{attribute 'qualified_only'}
VAR_GLOBAL CONSTANT
    DP_ID_DEFAULT_DATATYPE                   : UINT := 16#0000;
    DP_ID_PP_EMERGENCY_2                     : UINT := 16#0003;
    DP_ID_PP_EMERGENCY_1                     : UINT := 16#0004;

    DP_ID_DEBUG                              : UINT := 16#0069;
    DP_ID_MAIN_PCB_BOOT                      : UINT := 16#0070;

    DP_ID_COMMAND_HASH                       : UINT := 16#0167;
    DP_ID_DATA_HASH                          : UINT := 16#0169;
    DP_ID_VALUE_ERROR                        : UINT := 16#016A;
    DP_ID_VALUE_WARNING                      : UINT := 16#016B;
    DP_ID_VALUE_CAUSED_BRAKING               : UINT := 16#016C;
    DP_ID_LOCALISATION_HEARTBEAT             : UINT := 16#016E;
    DP_ID_SENSOR_HUB_HEARTBEAT               : UINT := 16#016F;
    DP_ID_FRONTEND_HEARTBEATING              : UINT := 16#0170;
    DP_ID_CONFIG_HASH                        : UINT := 16#0171;

    DP_ID_HV_V_LOW                           : UINT := 16#019D;   // critical
    DP_ID_BMS_TEMPERATURE_LOW                : UINT := 16#019E;

    DP_ID_FSM_STATE                          : UINT := 16#0202;
    DP_ID_FSM_TRANSITION_FAIL                : UINT := 16#0204;
    DP_ID_EMERGENCY                          : UINT := 16#0205;

    DP_ID_LEVI_SYSTEM_CHECK_SUCCESS          : UINT := 16#0220;
    DP_ID_LEVI_SYSTEM_CHECK_FAILURE          : UINT := 16#0221;
    DP_ID_PROP_1_SYSTEM_CHECK_SUCCESS        : UINT := 16#0222;
    DP_ID_PROP_1_SYSTEM_CHECK_FAILURE        : UINT := 16#0223;
    DP_ID_PROP_2_SYSTEM_CHECK_SUCCESS        : UINT := 16#0224;
    DP_ID_PROP_2_SYSTEM_CHECK_FAILURE        : UINT := 16#0225;
    DP_ID_RESET_FSM                          : UINT := 16#0226;
    DP_ID_EMERGENCY_STALE_CRITICAL_DATA      : UINT := 16#0227;
    DP_ID_LOCALIZATION_LIMIT_REACHED         : UINT := 16#0228;

    DP_ID_POD_STATE                          : UINT := 16#0250;   // u16,  pod->gs,  critical
    DP_ID_EMERGENCY_REASON                   : UINT := 16#0251;   // u16,  bidir,  critical
    DP_ID_POD_STATE_COMMAND                  : UINT := 16#0252;   // u16,  gs->pod

    DP_ID_LOCALIZATION                       : UINT := 16#0321;   // f32,  mm,  pod->gs

    DP_ID_HV_V_HIGH                          : UINT := 16#03A1;   // critical
    DP_ID_BMS_TEMPERATURE_HIGH               : UINT := 16#03A2;
    DP_ID_HVAL_STATE                         : UINT := 16#03A4;
    DP_ID_VDC_LINK                           : UINT := 16#03A7;   // critical
    DP_ID_PTC_ERRORS                         : UINT := 16#03B1;

    DP_ID_TEMP_MOTOR_LEFT_0                  : UINT := 16#04B0;
    DP_ID_TEMP_MOTOR_LEFT_1                  : UINT := 16#04B1;
    DP_ID_TEMP_MOTOR_LEFT_2                  : UINT := 16#04B2;
    DP_ID_TEMP_MOTOR_LEFT_3                  : UINT := 16#04B3;
    DP_ID_TEMP_MOTOR_LEFT_4                  : UINT := 16#04B4;
    DP_ID_TEMP_MOTOR_LEFT_5                  : UINT := 16#04B5;
    DP_ID_WORD_2                             : UINT := 16#04B6;   // critical
    DP_ID_IBUS_1                             : UINT := 16#04C2;
    DP_ID_IBUS_2                             : UINT := 16#04C6;

    DP_ID_PP_INIT_FAULT_1                    : UINT := 16#0507;
    DP_ID_PP_INIT_FAULT_2                    : UINT := 16#0508;
    DP_ID_TEMP_MOTOR_RIGHT_1                 : UINT := 16#050A;
    DP_ID_TEMP_MOTOR_RIGHT_2                 : UINT := 16#050B;
    DP_ID_TEMP_MOTOR_RIGHT_3                 : UINT := 16#050C;
    DP_ID_TEMP_MOTOR_RIGHT_4                 : UINT := 16#050D;
    DP_ID_TEMP_MOTOR_RIGHT_5                 : UINT := 16#050E;
    DP_ID_TEMP_MOTOR_RIGHT_6                 : UINT := 16#050F;

    DP_ID_TEMP_MOTOR_RIGHT_0                 : UINT := 16#0520;
    DP_ID_VELOCITY                           : UINT := 16#0527;   // i16,  mm/s,  pod->gs
    DP_ID_ROLL                               : UINT := 16#052E;
    DP_ID_PITCH                              : UINT := 16#052F;
    DP_ID_YAW                                : UINT := 16#0530;
    DP_ID_TEMP_HEMS1                         : UINT := 16#053C;
    DP_ID_TEMP_HEMS2                         : UINT := 16#053D;
    DP_ID_TEMP_HEMS3                         : UINT := 16#053E;
    DP_ID_TEMP_HEMS4                         : UINT := 16#053F;
    DP_ID_TEMP_HEMS5                         : UINT := 16#0540;
    DP_ID_TEMP_HEMS6                         : UINT := 16#0541;
    DP_ID_TEMP_HEMS7                         : UINT := 16#0542;
    DP_ID_TEMP_HEMS8                         : UINT := 16#0543;
    DP_ID_TEMP_EMS1                          : UINT := 16#0544;
    DP_ID_TEMP_EMS2                          : UINT := 16#0545;
    DP_ID_TEMP_EMS3                          : UINT := 16#0546;
    DP_ID_TEMP_EMS4                          : UINT := 16#0547;
    DP_ID_TEMP_EMS5                          : UINT := 16#0548;
    DP_ID_TEMP_EMS6                          : UINT := 16#0549;
    DP_ID_TEMP_EMS7                          : UINT := 16#054A;
    DP_ID_TEMP_EMS8                          : UINT := 16#054B;
    DP_ID_TEMP_MOTOR_RIGHT_7                 : UINT := 16#0555;
    DP_ID_TEMP_MOTOR_LEFT_6                  : UINT := 16#0556;
    DP_ID_TEMP_MOTOR_LEFT_7                  : UINT := 16#0557;
    DP_ID_LEVI_HEARTBEAT                     : UINT := 16#0567;   // critical
    DP_ID_LEVI_FAULT                         : UINT := 16#0568;

    DP_ID_WORD_1                             : UINT := 16#05B8;   // critical

    DP_ID_ISOLATION_RESISTANCE               : UINT := 16#0610;   // critical
    DP_ID_BUS_CURRENT                        : UINT := 16#0611;   // critical

    DP_ID_PRESSURE_LOW                       : UINT := 16#0666;   // critical
    DP_ID_PRESSURE_HIGH                      : UINT := 16#0667;   // critical

    DP_ID_SENSOR_HUB_EMERGENCY               : UINT := 16#0696;
    DP_ID_PTC_ERROR_EMERGENCY                : UINT := 16#0697;
    DP_ID_BMS_ERROR_LOW_VOLTAGE              : UINT := 16#0698;
    DP_ID_BMS_ERROR_HIGH_VOLTAGE             : UINT := 16#0699;

    DP_ID_LEVI_FAULT_DRIVE_NUMBER            : UINT := 16#0777;

    DP_ID_OFFSET_1                           : UINT := 16#0848;   // f32,  mm,  pod->gs
    DP_ID_OFFSET_2                           : UINT := 16#0849;   // f32,  mm,  pod->gs
    DP_ID_OFFSET_3                           : UINT := 16#084A;   // f32,  mm,  pod->gs
    DP_ID_OFFSET_4                           : UINT := 16#084B;   // f32,  mm,  pod->gs
    DP_ID_OFFSET_5                           : UINT := 16#084C;   // f32,  mm,  pod->gs
    DP_ID_OFFSET_6                           : UINT := 16#084D;   // f32,  mm,  pod->gs

    DP_ID_BARCODE_POSITION                   : UINT := 16#0900;
    DP_ID_BARCODE_VELOCITY                   : UINT := 16#0901;
    DP_ID_BARCODE_ID                         : UINT := 16#0902;
    DP_ID_BARCODE_QUALITY                    : UINT := 16#0903;
    DP_ID_LEVI_STATE                         : UINT := 16#0904;   // i16,  pod->gs,  critical
    DP_ID_LEVI_COMMAND                       : UINT := 16#0905;   // i16,  bidir,  critical
    DP_ID_LEVI_READY                         : UINT := 16#0906;   // u8,  pod->gs
    DP_ID_LEVI_Z_TARGET                      : UINT := 16#0907;   // f64,  m,  pod->gs
    DP_ID_LEVI_PITCH_TARGET                  : UINT := 16#0908;   // f64,  rad,  pod->gs
    DP_ID_LEVI_ROLL_TARGET                   : UINT := 16#0909;   // f64,  rad,  pod->gs
    DP_ID_LEVI_Y_TARGET_AIRGAP               : UINT := 16#090A;   // f64,  m,  pod->gs
    DP_ID_LEVI_YAW_TARGET                    : UINT := 16#090B;   // f64,  rad,  pod->gs
    DP_ID_LEVI_Z_LIFTOFF                     : UINT := 16#090C;   // f64,  m,  pod->gs
    DP_ID_LEVI_Z                             : UINT := 16#090D;   // f64,  m,  pod->gs,  critical
    DP_ID_LEVI_ROLL                          : UINT := 16#090E;   // f64,  rad,  pod->gs,  critical
    DP_ID_LEVI_PITCH                         : UINT := 16#090F;   // f64,  rad,  pod->gs,  critical
    DP_ID_LEVI_Y                             : UINT := 16#0910;   // f64,  m,  pod->gs,  critical
    DP_ID_LEVI_YAW                           : UINT := 16#0911;   // f64,  rad,  pod->gs,  critical
    DP_ID_LEVI_RESET_BUSY                    : UINT := 16#0912;   // u8,  pod->gs
    DP_ID_LEVI_RESET_ERROR                   : UINT := 16#0913;   // u8,  pod->gs
    DP_ID_LEVI_DRIVE_ERROR                   : UINT := 16#0914;   // u8,  pod->gs,  critical
    DP_ID_LEVI_N_DRIVE_WARNINGS              : UINT := 16#0915;   // u16,  pod->gs
    DP_ID_LEVI_N_DRIVE_ERRORS                : UINT := 16#0916;   // u16,  pod->gs
    DP_ID_LEVI_ERROR_RESETTABLE              : UINT := 16#0917;   // u8,  pod->gs,  critical
    DP_ID_LEVI_ERROR_EMERGENCY               : UINT := 16#0918;   // u8,  pod->gs,  critical
    DP_ID_LEVI_ERROR_NON_EMERGENCY           : UINT := 16#0919;   // u8,  pod->gs,  critical
    DP_ID_LEVI_ALL_DRIVES_HIGH_VOLTAGE       : UINT := 16#091A;   // u8,  pod->gs
    DP_ID_LEVI_N_VERTICAL_SENSORS_REJECTED   : UINT := 16#091B;   // u16,  pod->gs
    DP_ID_LEVI_N_LATERAL_SENSORS_REJECTED    : UINT := 16#091C;   // u16,  pod->gs
    DP_ID_LEVI_SENSOR_DATA_0                 : UINT := 16#091D;   // f64,  mm,  pod->gs
    DP_ID_LEVI_SENSOR_DATA_1                 : UINT := 16#091E;   // f64,  mm,  pod->gs
    DP_ID_LEVI_SENSOR_DATA_2                 : UINT := 16#091F;   // f64,  mm,  pod->gs
    DP_ID_LEVI_SENSOR_DATA_3                 : UINT := 16#0920;   // f64,  mm,  pod->gs
    DP_ID_LEVI_SENSOR_DATA_4                 : UINT := 16#0921;   // f64,  mm,  pod->gs
    DP_ID_LEVI_SENSOR_DATA_5                 : UINT := 16#0922;   // f64,  mm,  pod->gs
    DP_ID_LEVI_SENSOR_DATA_6                 : UINT := 16#0923;   // f64,  mm,  pod->gs
    DP_ID_LEVI_SENSOR_DATA_7                 : UINT := 16#0924;   // f64,  mm,  pod->gs
    DP_ID_LEVI_SENSOR_DATA_8                 : UINT := 16#0925;   // f64,  mm,  pod->gs
    DP_ID_LEVI_SENSOR_DATA_9                 : UINT := 16#0926;   // f64,  mm,  pod->gs
    DP_ID_LEVI_SENSOR_DATA_10                : UINT := 16#0927;   // f64,  mm,  pod->gs
    DP_ID_LEVI_SENSOR_DATA_11                : UINT := 16#0928;   // f64,  mm,  pod->gs
    DP_ID_LEVI_DRIVE_STATUS_0                : UINT := 16#0929;   // u16,  pod->gs
    DP_ID_LEVI_DRIVE_STATUS_1                : UINT := 16#092A;   // u16,  pod->gs
    DP_ID_LEVI_DRIVE_STATUS_2                : UINT := 16#092B;   // u16,  pod->gs
    DP_ID_LEVI_DRIVE_STATUS_3                : UINT := 16#092C;   // u16,  pod->gs
    DP_ID_LEVI_DRIVE_STATUS_4                : UINT := 16#092D;   // u16,  pod->gs
    DP_ID_LEVI_DRIVE_STATUS_5                : UINT := 16#092E;   // u16,  pod->gs
    DP_ID_LEVI_DRIVE_STATUS_6                : UINT := 16#092F;   // u16,  pod->gs
    DP_ID_LEVI_DRIVE_STATUS_7                : UINT := 16#0930;   // u16,  pod->gs
    DP_ID_LEVI_DRIVE_STATUS_8                : UINT := 16#0931;   // u16,  pod->gs
    DP_ID_LEVI_DRIVE_STATUS_9                : UINT := 16#0932;   // u16,  pod->gs
    DP_ID_LEVI_DRIVE_STATUS_10               : UINT := 16#0933;   // u16,  pod->gs
    DP_ID_LEVI_DRIVE_STATUS_11               : UINT := 16#0934;   // u16,  pod->gs
    DP_ID_LEVI_DRIVE_STATUS_12               : UINT := 16#0935;   // u16,  pod->gs
    DP_ID_LEVI_DRIVE_STATUS_13               : UINT := 16#0936;   // u16,  pod->gs
    DP_ID_LEVI_DRIVE_STATUS_14               : UINT := 16#0937;   // u16,  pod->gs
    DP_ID_LEVI_DRIVE_STATUS_15               : UINT := 16#0938;   // u16,  pod->gs
    DP_ID_LEVI_DRIVE_STATUS_16               : UINT := 16#0939;   // u16,  pod->gs
    DP_ID_LEVI_DRIVE_STATUS_17               : UINT := 16#093A;   // u16,  pod->gs
    DP_ID_LEVI_DRIVE_STATUS_18               : UINT := 16#093B;   // u16,  pod->gs
    DP_ID_LEVI_DRIVE_STATUS_19               : UINT := 16#093C;   // u16,  pod->gs
    DP_ID_LEVI_DRIVE_STATUS_20               : UINT := 16#093D;   // u16,  pod->gs
    DP_ID_LEVI_DRIVE_STATUS_21               : UINT := 16#093E;   // u16,  pod->gs
    DP_ID_LEVI_DRIVE_STATUS_22               : UINT := 16#093F;   // u16,  pod->gs
    DP_ID_LEVI_DRIVE_STATUS_23               : UINT := 16#0940;   // u16,  pod->gs
    DP_ID_LEVI_DRIVE_DIAGNOSTICS_0           : UINT := 16#0941;   // u16,  pod->gs
    DP_ID_LEVI_DRIVE_DIAGNOSTICS_1           : UINT := 16#0942;   // u16,  pod->gs
    DP_ID_LEVI_DRIVE_DIAGNOSTICS_2           : UINT := 16#0943;   // u16,  pod->gs
    DP_ID_LEVI_DRIVE_DIAGNOSTICS_3           : UINT := 16#0944;   // u16,  pod->gs
    DP_ID_LEVI_DRIVE_DIAGNOSTICS_4           : UINT := 16#0945;   // u16,  pod->gs
    DP_ID_LEVI_DRIVE_DIAGNOSTICS_5           : UINT := 16#0946;   // u16,  pod->gs
    DP_ID_LEVI_DRIVE_DIAGNOSTICS_6           : UINT := 16#0947;   // u16,  pod->gs
    DP_ID_LEVI_DRIVE_DIAGNOSTICS_7           : UINT := 16#0948;   // u16,  pod->gs
    DP_ID_LEVI_DRIVE_DIAGNOSTICS_8           : UINT := 16#0949;   // u16,  pod->gs
    DP_ID_LEVI_DRIVE_DIAGNOSTICS_9           : UINT := 16#094A;   // u16,  pod->gs
    DP_ID_LEVI_DRIVE_DIAGNOSTICS_10          : UINT := 16#094B;   // u16,  pod->gs
    DP_ID_LEVI_DRIVE_DIAGNOSTICS_11          : UINT := 16#094C;   // u16,  pod->gs
    DP_ID_LEVI_DRIVE_DIAGNOSTICS_12          : UINT := 16#094D;   // u16,  pod->gs
    DP_ID_LEVI_DRIVE_DIAGNOSTICS_13          : UINT := 16#094E;   // u16,  pod->gs
    DP_ID_LEVI_DRIVE_DIAGNOSTICS_14          : UINT := 16#094F;   // u16,  pod->gs
    DP_ID_LEVI_DRIVE_DIAGNOSTICS_15          : UINT := 16#0950;   // u16,  pod->gs
    DP_ID_LEVI_DRIVE_DIAGNOSTICS_16          : UINT := 16#0951;   // u16,  pod->gs
    DP_ID_LEVI_DRIVE_DIAGNOSTICS_17          : UINT := 16#0952;   // u16,  pod->gs
    DP_ID_LEVI_DRIVE_DIAGNOSTICS_18          : UINT := 16#0953;   // u16,  pod->gs
    DP_ID_LEVI_DRIVE_DIAGNOSTICS_19          : UINT := 16#0954;   // u16,  pod->gs
    DP_ID_LEVI_DRIVE_DIAGNOSTICS_20          : UINT := 16#0955;   // u16,  pod->gs
    DP_ID_LEVI_DRIVE_DIAGNOSTICS_21          : UINT := 16#0956;   // u16,  pod->gs
    DP_ID_LEVI_DRIVE_DIAGNOSTICS_22          : UINT := 16#0957;   // u16,  pod->gs
    DP_ID_LEVI_DRIVE_DIAGNOSTICS_23          : UINT := 16#0958;   // u16,  pod->gs
    DP_ID_LEVI_REAL_CURRENTS_0               : UINT := 16#0959;   // f64,  A,  pod->gs,  critical
    DP_ID_LEVI_REAL_CURRENTS_1               : UINT := 16#095A;   // f64,  A,  pod->gs,  critical
    DP_ID_LEVI_REAL_CURRENTS_2               : UINT := 16#095B;   // f64,  A,  pod->gs,  critical
    DP_ID_LEVI_REAL_CURRENTS_3               : UINT := 16#095C;   // f64,  A,  pod->gs,  critical
    DP_ID_LEVI_REAL_CURRENTS_4               : UINT := 16#095D;   // f64,  A,  pod->gs,  critical
    DP_ID_LEVI_REAL_CURRENTS_5               : UINT := 16#095E;   // f64,  A,  pod->gs,  critical
    DP_ID_LEVI_REAL_CURRENTS_6               : UINT := 16#095F;   // f64,  A,  pod->gs,  critical
    DP_ID_LEVI_REAL_CURRENTS_7               : UINT := 16#0960;   // f64,  A,  pod->gs,  critical
    DP_ID_LEVI_REAL_CURRENTS_8               : UINT := 16#0961;   // f64,  A,  pod->gs,  critical
    DP_ID_LEVI_REAL_CURRENTS_9               : UINT := 16#0962;   // f64,  A,  pod->gs,  critical
    DP_ID_LEVI_REAL_CURRENTS_10              : UINT := 16#0963;   // f64,  A,  pod->gs,  critical
    DP_ID_LEVI_REAL_CURRENTS_11              : UINT := 16#0964;   // f64,  A,  pod->gs,  critical
    DP_ID_LEVI_REAL_CURRENTS_12              : UINT := 16#0965;   // f64,  A,  pod->gs,  critical
    DP_ID_LEVI_REAL_CURRENTS_13              : UINT := 16#0966;   // f64,  A,  pod->gs,  critical
    DP_ID_LEVI_REAL_CURRENTS_14              : UINT := 16#0967;   // f64,  A,  pod->gs,  critical
    DP_ID_LEVI_REAL_CURRENTS_15              : UINT := 16#0968;   // f64,  A,  pod->gs,  critical
    DP_ID_LEVI_REAL_CURRENTS_16              : UINT := 16#0969;   // f64,  A,  pod->gs,  critical
    DP_ID_LEVI_REAL_CURRENTS_17              : UINT := 16#096A;   // f64,  A,  pod->gs,  critical
    DP_ID_LEVI_REAL_CURRENTS_18              : UINT := 16#096B;   // f64,  A,  pod->gs,  critical
    DP_ID_LEVI_REAL_CURRENTS_19              : UINT := 16#096C;   // f64,  A,  pod->gs,  critical
    DP_ID_LEVI_REAL_CURRENTS_20              : UINT := 16#096D;   // f64,  A,  pod->gs,  critical
    DP_ID_LEVI_REAL_CURRENTS_21              : UINT := 16#096E;   // f64,  A,  pod->gs,  critical
    DP_ID_LEVI_REAL_CURRENTS_22              : UINT := 16#096F;   // f64,  A,  pod->gs,  critical
    DP_ID_LEVI_REAL_CURRENTS_23              : UINT := 16#0970;   // f64,  A,  pod->gs,  critical
    DP_ID_LEVI_DC_BUS_VOLTAGE_0              : UINT := 16#0971;   // u16,  V,  pod->gs,  critical
    DP_ID_LEVI_DC_BUS_VOLTAGE_1              : UINT := 16#0972;   // u16,  V,  pod->gs,  critical
    DP_ID_LEVI_DC_BUS_VOLTAGE_2              : UINT := 16#0973;   // u16,  V,  pod->gs,  critical
    DP_ID_LEVI_DC_BUS_VOLTAGE_3              : UINT := 16#0974;   // u16,  V,  pod->gs,  critical
    DP_ID_LEVI_DC_BUS_VOLTAGE_4              : UINT := 16#0975;   // u16,  V,  pod->gs,  critical
    DP_ID_LEVI_DC_BUS_VOLTAGE_5              : UINT := 16#0976;   // u16,  V,  pod->gs,  critical
    DP_ID_LEVI_DC_BUS_VOLTAGE_6              : UINT := 16#0977;   // u16,  V,  pod->gs,  critical
    DP_ID_LEVI_DC_BUS_VOLTAGE_7              : UINT := 16#0978;   // u16,  V,  pod->gs,  critical
    DP_ID_LEVI_DC_BUS_VOLTAGE_8              : UINT := 16#0979;   // u16,  V,  pod->gs,  critical
    DP_ID_LEVI_DC_BUS_VOLTAGE_9              : UINT := 16#097A;   // u16,  V,  pod->gs,  critical
    DP_ID_LEVI_DC_BUS_VOLTAGE_10             : UINT := 16#097B;   // u16,  V,  pod->gs,  critical
    DP_ID_LEVI_DC_BUS_VOLTAGE_11             : UINT := 16#097C;   // u16,  V,  pod->gs,  critical
    DP_ID_LEVI_DC_BUS_VOLTAGE_12             : UINT := 16#097D;   // u16,  V,  pod->gs,  critical
    DP_ID_LEVI_DC_BUS_VOLTAGE_13             : UINT := 16#097E;   // u16,  V,  pod->gs,  critical
    DP_ID_LEVI_DC_BUS_VOLTAGE_14             : UINT := 16#097F;   // u16,  V,  pod->gs,  critical
    DP_ID_LEVI_DC_BUS_VOLTAGE_15             : UINT := 16#0980;   // u16,  V,  pod->gs,  critical
    DP_ID_LEVI_DC_BUS_VOLTAGE_16             : UINT := 16#0981;   // u16,  V,  pod->gs,  critical
    DP_ID_LEVI_DC_BUS_VOLTAGE_17             : UINT := 16#0982;   // u16,  V,  pod->gs,  critical
    DP_ID_LEVI_DC_BUS_VOLTAGE_18             : UINT := 16#0983;   // u16,  V,  pod->gs,  critical
    DP_ID_LEVI_DC_BUS_VOLTAGE_19             : UINT := 16#0984;   // u16,  V,  pod->gs,  critical
    DP_ID_LEVI_DC_BUS_VOLTAGE_20             : UINT := 16#0985;   // u16,  V,  pod->gs,  critical
    DP_ID_LEVI_DC_BUS_VOLTAGE_21             : UINT := 16#0986;   // u16,  V,  pod->gs,  critical
    DP_ID_LEVI_DC_BUS_VOLTAGE_22             : UINT := 16#0987;   // u16,  V,  pod->gs,  critical
    DP_ID_LEVI_DC_BUS_VOLTAGE_23             : UINT := 16#0988;   // u16,  V,  pod->gs,  critical
    DP_ID_LEVI_PERIPHERY_VOLTAGE_0           : UINT := 16#0989;   // u16,  V,  pod->gs
    DP_ID_LEVI_PERIPHERY_VOLTAGE_1           : UINT := 16#098A;   // u16,  V,  pod->gs
    DP_ID_LEVI_PERIPHERY_VOLTAGE_2           : UINT := 16#098B;   // u16,  V,  pod->gs
    DP_ID_LEVI_PERIPHERY_VOLTAGE_3           : UINT := 16#098C;   // u16,  V,  pod->gs
    DP_ID_LEVI_PERIPHERY_VOLTAGE_4           : UINT := 16#098D;   // u16,  V,  pod->gs
    DP_ID_LEVI_PERIPHERY_VOLTAGE_5           : UINT := 16#098E;   // u16,  V,  pod->gs
    DP_ID_LEVI_PERIPHERY_VOLTAGE_6           : UINT := 16#098F;   // u16,  V,  pod->gs
    DP_ID_LEVI_PERIPHERY_VOLTAGE_7           : UINT := 16#0990;   // u16,  V,  pod->gs
    DP_ID_LEVI_PERIPHERY_VOLTAGE_8           : UINT := 16#0991;   // u16,  V,  pod->gs
    DP_ID_LEVI_PERIPHERY_VOLTAGE_9           : UINT := 16#0992;   // u16,  V,  pod->gs
    DP_ID_LEVI_PERIPHERY_VOLTAGE_10          : UINT := 16#0993;   // u16,  V,  pod->gs
    DP_ID_LEVI_PERIPHERY_VOLTAGE_11          : UINT := 16#0994;   // u16,  V,  pod->gs
    DP_ID_LEVI_PERIPHERY_VOLTAGE_12          : UINT := 16#0995;   // u16,  V,  pod->gs
    DP_ID_LEVI_PERIPHERY_VOLTAGE_13          : UINT := 16#0996;   // u16,  V,  pod->gs
    DP_ID_LEVI_PERIPHERY_VOLTAGE_14          : UINT := 16#0997;   // u16,  V,  pod->gs
    DP_ID_LEVI_PERIPHERY_VOLTAGE_15          : UINT := 16#0998;   // u16,  V,  pod->gs
    DP_ID_LEVI_PERIPHERY_VOLTAGE_16          : UINT := 16#0999;   // u16,  V,  pod->gs
    DP_ID_LEVI_PERIPHERY_VOLTAGE_17          : UINT := 16#099A;   // u16,  V,  pod->gs
    DP_ID_LEVI_PERIPHERY_VOLTAGE_18          : UINT := 16#099B;   // u16,  V,  pod->gs
    DP_ID_LEVI_PERIPHERY_VOLTAGE_19          : UINT := 16#099C;   // u16,  V,  pod->gs
    DP_ID_LEVI_PERIPHERY_VOLTAGE_20          : UINT := 16#099D;   // u16,  V,  pod->gs
    DP_ID_LEVI_PERIPHERY_VOLTAGE_21          : UINT := 16#099E;   // u16,  V,  pod->gs
    DP_ID_LEVI_PERIPHERY_VOLTAGE_22          : UINT := 16#099F;   // u16,  V,  pod->gs
    DP_ID_LEVI_PERIPHERY_VOLTAGE_23          : UINT := 16#09A0;   // u16,  V,  pod->gs
    DP_ID_LEVI_REQUESTED_CURRENTS_0          : UINT := 16#09A1;   // f64,  A,  pod->gs
    DP_ID_LEVI_REQUESTED_CURRENTS_1          : UINT := 16#09A2;   // f64,  A,  pod->gs
    DP_ID_LEVI_REQUESTED_CURRENTS_2          : UINT := 16#09A3;   // f64,  A,  pod->gs
    DP_ID_LEVI_REQUESTED_CURRENTS_3          : UINT := 16#09A4;   // f64,  A,  pod->gs
    DP_ID_LEVI_REQUESTED_CURRENTS_4          : UINT := 16#09A5;   // f64,  A,  pod->gs
    DP_ID_LEVI_REQUESTED_CURRENTS_5          : UINT := 16#09A6;   // f64,  A,  pod->gs
    DP_ID_LEVI_REQUESTED_CURRENTS_6          : UINT := 16#09A7;   // f64,  A,  pod->gs
    DP_ID_LEVI_REQUESTED_CURRENTS_7          : UINT := 16#09A8;   // f64,  A,  pod->gs
    DP_ID_LEVI_REQUESTED_CURRENTS_8          : UINT := 16#09A9;   // f64,  A,  pod->gs
    DP_ID_LEVI_REQUESTED_CURRENTS_9          : UINT := 16#09AA;   // f64,  A,  pod->gs
    DP_ID_LEVI_REQUESTED_CURRENTS_10         : UINT := 16#09AB;   // f64,  A,  pod->gs
    DP_ID_LEVI_REQUESTED_CURRENTS_11         : UINT := 16#09AC;   // f64,  A,  pod->gs
    DP_ID_LEVI_CONTROL_WORD_0                : UINT := 16#09AD;   // u16,  pod->gs
    DP_ID_LEVI_CONTROL_WORD_1                : UINT := 16#09AE;   // u16,  pod->gs
    DP_ID_LEVI_CONTROL_WORD_2                : UINT := 16#09AF;   // u16,  pod->gs
    DP_ID_LEVI_CONTROL_WORD_3                : UINT := 16#09B0;   // u16,  pod->gs
    DP_ID_LEVI_CONTROL_WORD_4                : UINT := 16#09B1;   // u16,  pod->gs
    DP_ID_LEVI_CONTROL_WORD_5                : UINT := 16#09B2;   // u16,  pod->gs
    DP_ID_LEVI_CONTROL_WORD_6                : UINT := 16#09B3;   // u16,  pod->gs
    DP_ID_LEVI_CONTROL_WORD_7                : UINT := 16#09B4;   // u16,  pod->gs
    DP_ID_LEVI_CONTROL_WORD_8                : UINT := 16#09B5;   // u16,  pod->gs
    DP_ID_LEVI_CONTROL_WORD_9                : UINT := 16#09B6;   // u16,  pod->gs
    DP_ID_LEVI_CONTROL_WORD_10               : UINT := 16#09B7;   // u16,  pod->gs
    DP_ID_LEVI_CONTROL_WORD_11               : UINT := 16#09B8;   // u16,  pod->gs
    DP_ID_LEVI_CONTROL_WORD_12               : UINT := 16#09B9;   // u16,  pod->gs
    DP_ID_LEVI_CONTROL_WORD_13               : UINT := 16#09BA;   // u16,  pod->gs
    DP_ID_LEVI_CONTROL_WORD_14               : UINT := 16#09BB;   // u16,  pod->gs
    DP_ID_LEVI_CONTROL_WORD_15               : UINT := 16#09BC;   // u16,  pod->gs
    DP_ID_LEVI_CONTROL_WORD_16               : UINT := 16#09BD;   // u16,  pod->gs
    DP_ID_LEVI_CONTROL_WORD_17               : UINT := 16#09BE;   // u16,  pod->gs
    DP_ID_LEVI_CONTROL_WORD_18               : UINT := 16#09BF;   // u16,  pod->gs
    DP_ID_LEVI_CONTROL_WORD_19               : UINT := 16#09C0;   // u16,  pod->gs
    DP_ID_LEVI_CONTROL_WORD_20               : UINT := 16#09C1;   // u16,  pod->gs
    DP_ID_LEVI_CONTROL_WORD_21               : UINT := 16#09C2;   // u16,  pod->gs
    DP_ID_LEVI_CONTROL_WORD_22               : UINT := 16#09C3;   // u16,  pod->gs
    DP_ID_LEVI_CONTROL_WORD_23               : UINT := 16#09C4;   // u16,  pod->gs
    DP_ID_LEVI_ERROR_SPECIFICS_0             : UINT := 16#09C5;   // i8,  pod->gs,  critical
    DP_ID_LEVI_ERROR_SPECIFICS_1             : UINT := 16#09C6;   // i8,  pod->gs,  critical
    DP_ID_LEVI_ERROR_SPECIFICS_2             : UINT := 16#09C7;   // i8,  pod->gs,  critical
    DP_ID_LEVI_ERROR_SPECIFICS_3             : UINT := 16#09C8;   // i8,  pod->gs,  critical
    DP_ID_LEVI_ERROR_SPECIFICS_4             : UINT := 16#09C9;   // i8,  pod->gs,  critical
    DP_ID_LEVI_ERROR_SPECIFICS_5             : UINT := 16#09CA;   // i8,  pod->gs,  critical
    DP_ID_LEVI_ERROR_SPECIFICS_6             : UINT := 16#09CB;   // i8,  pod->gs,  critical
    DP_ID_LEVI_ERROR_SPECIFICS_7             : UINT := 16#09CC;   // i8,  pod->gs,  critical
    DP_ID_LEVI_ERROR_SPECIFICS_8             : UINT := 16#09CD;   // i8,  pod->gs,  critical
    DP_ID_LEVI_ERROR_SPECIFICS_9             : UINT := 16#09CE;   // i8,  pod->gs,  critical
    DP_ID_LEVI_ERROR_SPECIFICS_10            : UINT := 16#09CF;   // i8,  pod->gs,  critical
    DP_ID_LEVI_ERROR_SPECIFICS_11            : UINT := 16#09D0;   // i8,  pod->gs,  critical
    DP_ID_LEVI_ERROR_SPECIFICS_12            : UINT := 16#09D1;   // i8,  pod->gs,  critical
    DP_ID_LEVI_ERROR_SPECIFICS_13            : UINT := 16#09D2;   // i8,  pod->gs,  critical
    DP_ID_LEVI_ERROR_SPECIFICS_14            : UINT := 16#09D3;   // i8,  pod->gs,  critical
    DP_ID_LEVI_ERROR_SPECIFICS_15            : UINT := 16#09D4;   // i8,  pod->gs,  critical
    DP_ID_LEVI_ERROR_SPECIFICS_16            : UINT := 16#09D5;   // i8,  pod->gs,  critical
    DP_ID_LEVI_ERROR_SPECIFICS_17            : UINT := 16#09D6;   // i8,  pod->gs,  critical
    DP_ID_LEVI_ERROR_SPECIFICS_18            : UINT := 16#09D7;   // i8,  pod->gs,  critical
    DP_ID_LEVI_ERROR_SPECIFICS_19            : UINT := 16#09D8;   // i8,  pod->gs,  critical
    DP_ID_LEVI_ERROR_SPECIFICS_20            : UINT := 16#09D9;   // i8,  pod->gs,  critical
    DP_ID_LEVI_ERROR_SPECIFICS_21            : UINT := 16#09DA;   // i8,  pod->gs,  critical
    DP_ID_LEVI_ERROR_SPECIFICS_22            : UINT := 16#09DB;   // i8,  pod->gs,  critical
    DP_ID_LEVI_ERROR_SPECIFICS_23            : UINT := 16#09DC;   // i8,  pod->gs,  critical
    DP_ID_LEVI_DRIVE_FEEDBACK_TIMEOUTS_0     : UINT := 16#09DD;   // u16,  pod->gs
    DP_ID_LEVI_DRIVE_FEEDBACK_TIMEOUTS_1     : UINT := 16#09DE;   // u16,  pod->gs
    DP_ID_LEVI_DRIVE_FEEDBACK_TIMEOUTS_2     : UINT := 16#09DF;   // u16,  pod->gs
    DP_ID_LEVI_DRIVE_FEEDBACK_TIMEOUTS_3     : UINT := 16#09E0;   // u16,  pod->gs
    DP_ID_LEVI_DRIVE_FEEDBACK_TIMEOUTS_4     : UINT := 16#09E1;   // u16,  pod->gs
    DP_ID_LEVI_DRIVE_FEEDBACK_TIMEOUTS_5     : UINT := 16#09E2;   // u16,  pod->gs
    DP_ID_LEVI_DRIVE_FEEDBACK_TIMEOUTS_6     : UINT := 16#09E3;   // u16,  pod->gs
    DP_ID_LEVI_DRIVE_FEEDBACK_TIMEOUTS_7     : UINT := 16#09E4;   // u16,  pod->gs
    DP_ID_LEVI_DRIVE_FEEDBACK_TIMEOUTS_8     : UINT := 16#09E5;   // u16,  pod->gs
    DP_ID_LEVI_DRIVE_FEEDBACK_TIMEOUTS_9     : UINT := 16#09E6;   // u16,  pod->gs
    DP_ID_LEVI_DRIVE_FEEDBACK_TIMEOUTS_10    : UINT := 16#09E7;   // u16,  pod->gs
    DP_ID_LEVI_DRIVE_FEEDBACK_TIMEOUTS_11    : UINT := 16#09E8;   // u16,  pod->gs
    DP_ID_LEVI_DRIVE_FEEDBACK_TIMEOUTS_12    : UINT := 16#09E9;   // u16,  pod->gs
    DP_ID_LEVI_DRIVE_FEEDBACK_TIMEOUTS_13    : UINT := 16#09EA;   // u16,  pod->gs
    DP_ID_LEVI_DRIVE_FEEDBACK_TIMEOUTS_14    : UINT := 16#09EB;   // u16,  pod->gs
    DP_ID_LEVI_DRIVE_FEEDBACK_TIMEOUTS_15    : UINT := 16#09EC;   // u16,  pod->gs
    DP_ID_LEVI_DRIVE_FEEDBACK_TIMEOUTS_16    : UINT := 16#09ED;   // u16,  pod->gs
    DP_ID_LEVI_DRIVE_FEEDBACK_TIMEOUTS_17    : UINT := 16#09EE;   // u16,  pod->gs
    DP_ID_LEVI_DRIVE_FEEDBACK_TIMEOUTS_18    : UINT := 16#09EF;   // u16,  pod->gs
    DP_ID_LEVI_DRIVE_FEEDBACK_TIMEOUTS_19    : UINT := 16#09F0;   // u16,  pod->gs
    DP_ID_LEVI_DRIVE_FEEDBACK_TIMEOUTS_20    : UINT := 16#09F1;   // u16,  pod->gs
    DP_ID_LEVI_DRIVE_FEEDBACK_TIMEOUTS_21    : UINT := 16#09F2;   // u16,  pod->gs
    DP_ID_LEVI_DRIVE_FEEDBACK_TIMEOUTS_22    : UINT := 16#09F3;   // u16,  pod->gs
    DP_ID_LEVI_DRIVE_FEEDBACK_TIMEOUTS_23    : UINT := 16#09F4;   // u16,  pod->gs
    DP_ID_LEVI_DRIVE_CURRENT_ERROR_0         : UINT := 16#09F5;   // u8,  pod->gs,  critical
    DP_ID_LEVI_DRIVE_CURRENT_ERROR_1         : UINT := 16#09F6;   // u8,  pod->gs,  critical
    DP_ID_LEVI_DRIVE_CURRENT_ERROR_2         : UINT := 16#09F7;   // u8,  pod->gs,  critical
    DP_ID_LEVI_DRIVE_CURRENT_ERROR_3         : UINT := 16#09F8;   // u8,  pod->gs,  critical
    DP_ID_LEVI_DRIVE_CURRENT_ERROR_4         : UINT := 16#09F9;   // u8,  pod->gs,  critical
    DP_ID_LEVI_DRIVE_CURRENT_ERROR_5         : UINT := 16#09FA;   // u8,  pod->gs,  critical
    DP_ID_LEVI_DRIVE_CURRENT_ERROR_6         : UINT := 16#09FB;   // u8,  pod->gs,  critical
    DP_ID_LEVI_DRIVE_CURRENT_ERROR_7         : UINT := 16#09FC;   // u8,  pod->gs,  critical
    DP_ID_LEVI_DRIVE_CURRENT_ERROR_8         : UINT := 16#09FD;   // u8,  pod->gs,  critical
    DP_ID_LEVI_DRIVE_CURRENT_ERROR_9         : UINT := 16#09FE;   // u8,  pod->gs,  critical
    DP_ID_LEVI_DRIVE_CURRENT_ERROR_10        : UINT := 16#09FF;   // u8,  pod->gs,  critical
    DP_ID_LEVI_DRIVE_CURRENT_ERROR_11        : UINT := 16#0A00;   // u8,  pod->gs,  critical
    DP_ID_LEVI_DRIVE_CURRENT_ERROR_12        : UINT := 16#0A01;   // u8,  pod->gs,  critical
    DP_ID_LEVI_DRIVE_CURRENT_ERROR_13        : UINT := 16#0A02;   // u8,  pod->gs,  critical
    DP_ID_LEVI_DRIVE_CURRENT_ERROR_14        : UINT := 16#0A03;   // u8,  pod->gs,  critical
    DP_ID_LEVI_DRIVE_CURRENT_ERROR_15        : UINT := 16#0A04;   // u8,  pod->gs,  critical
    DP_ID_LEVI_DRIVE_CURRENT_ERROR_16        : UINT := 16#0A05;   // u8,  pod->gs,  critical
    DP_ID_LEVI_DRIVE_CURRENT_ERROR_17        : UINT := 16#0A06;   // u8,  pod->gs,  critical
    DP_ID_LEVI_DRIVE_CURRENT_ERROR_18        : UINT := 16#0A07;   // u8,  pod->gs,  critical
    DP_ID_LEVI_DRIVE_CURRENT_ERROR_19        : UINT := 16#0A08;   // u8,  pod->gs,  critical
    DP_ID_LEVI_DRIVE_CURRENT_ERROR_20        : UINT := 16#0A09;   // u8,  pod->gs,  critical
    DP_ID_LEVI_DRIVE_CURRENT_ERROR_21        : UINT := 16#0A0A;   // u8,  pod->gs,  critical
    DP_ID_LEVI_DRIVE_CURRENT_ERROR_22        : UINT := 16#0A0B;   // u8,  pod->gs,  critical
    DP_ID_LEVI_DRIVE_CURRENT_ERROR_23        : UINT := 16#0A0C;   // u8,  pod->gs,  critical
    DP_ID_LEVI_OFFSET_AIRGAPS_0              : UINT := 16#0A0D;   // f64,  m,  pod->gs
    DP_ID_LEVI_OFFSET_AIRGAPS_1              : UINT := 16#0A0E;   // f64,  m,  pod->gs
    DP_ID_LEVI_OFFSET_AIRGAPS_2              : UINT := 16#0A0F;   // f64,  m,  pod->gs
    DP_ID_LEVI_OFFSET_AIRGAPS_3              : UINT := 16#0A10;   // f64,  m,  pod->gs
    DP_ID_LEVI_OFFSET_AIRGAPS_4              : UINT := 16#0A11;   // f64,  m,  pod->gs
    DP_ID_LEVI_OFFSET_AIRGAPS_5              : UINT := 16#0A12;   // f64,  m,  pod->gs
    DP_ID_LEVI_OFFSET_AIRGAPS_6              : UINT := 16#0A13;   // f64,  m,  pod->gs
    DP_ID_LEVI_OFFSET_AIRGAPS_7              : UINT := 16#0A14;   // f64,  m,  pod->gs
    DP_ID_LEVI_OFFSET_AIRGAPS_8              : UINT := 16#0A15;   // f64,  m,  pod->gs
    DP_ID_LEVI_OFFSET_AIRGAPS_9              : UINT := 16#0A16;   // f64,  m,  pod->gs
    DP_ID_LEVI_OFFSET_AIRGAPS_10             : UINT := 16#0A17;   // f64,  m,  pod->gs
    DP_ID_LEVI_OFFSET_AIRGAPS_11             : UINT := 16#0A18;   // f64,  m,  pod->gs

    DP_ID_LEVI_OPERATIONAL                   : UINT := 16#0A30;   // u8,  bidir
    DP_ID_LEVI_VERTICAL_ON                   : UINT := 16#0A31;   // u8,  bidir
    DP_ID_LEVI_LATERAL_ON                    : UINT := 16#0A32;   // u8,  bidir
    DP_ID_LEVI_MOTOR_ON                      : UINT := 16#0A33;   // u8,  bidir
    DP_ID_LEVI_TOTAL_ON                      : UINT := 16#0A34;   // u8,  bidir
    DP_ID_LEVI_PITCH_ON                      : UINT := 16#0A35;   // u8,  bidir
    DP_ID_LEVI_ROLL_ON                       : UINT := 16#0A36;   // u8,  bidir
    DP_ID_LEVI_Y_ON                          : UINT := 16#0A37;   // u8,  bidir
    DP_ID_LEVI_YAW_ON                        : UINT := 16#0A38;   // u8,  bidir
    DP_ID_LEVI_ENABLE_MANUAL_Z_TARGET        : UINT := 16#0A39;   // u8,  bidir
    DP_ID_LEVI_KP_TOT                        : UINT := 16#0A40;   // f64,  bidir
    DP_ID_LEVI_KI_TOT                        : UINT := 16#0A41;   // f64,  bidir
    DP_ID_LEVI_KD_TOT                        : UINT := 16#0A42;   // f64,  bidir
    DP_ID_LEVI_KF_TOT                        : UINT := 16#0A43;   // f64,  bidir
    DP_ID_LEVI_KI_TOT_INITIAL                : UINT := 16#0A44;   // f64,  bidir
    DP_ID_LEVI_KP_PITCH                      : UINT := 16#0A45;   // f64,  bidir
    DP_ID_LEVI_KI_PITCH                      : UINT := 16#0A46;   // f64,  bidir
    DP_ID_LEVI_KD_PITCH                      : UINT := 16#0A47;   // f64,  bidir
    DP_ID_LEVI_KF_PITCH                      : UINT := 16#0A48;   // f64,  bidir
    DP_ID_LEVI_KI_PITCH_INITIAL              : UINT := 16#0A49;   // f64,  bidir
    DP_ID_LEVI_KP_ROLL                       : UINT := 16#0A4A;   // f64,  bidir
    DP_ID_LEVI_KI_ROLL                       : UINT := 16#0A4B;   // f64,  bidir
    DP_ID_LEVI_KD_ROLL                       : UINT := 16#0A4C;   // f64,  bidir
    DP_ID_LEVI_KF_ROLL                       : UINT := 16#0A4D;   // f64,  bidir
    DP_ID_LEVI_KI_ROLL_INITIAL               : UINT := 16#0A4E;   // f64,  bidir
    DP_ID_LEVI_KP_LAT                        : UINT := 16#0A4F;   // f64,  bidir
    DP_ID_LEVI_KI_LAT                        : UINT := 16#0A50;   // f64,  bidir
    DP_ID_LEVI_KD_LAT                        : UINT := 16#0A51;   // f64,  bidir
    DP_ID_LEVI_KF_LAT                        : UINT := 16#0A52;   // f64,  bidir
    DP_ID_LEVI_KI_LAT_INITIAL                : UINT := 16#0A53;   // f64,  bidir
    DP_ID_LEVI_KP_YAW                        : UINT := 16#0A54;   // f64,  bidir
    DP_ID_LEVI_KI_YAW                        : UINT := 16#0A55;   // f64,  bidir
    DP_ID_LEVI_KD_YAW                        : UINT := 16#0A56;   // f64,  bidir
    DP_ID_LEVI_KF_YAW                        : UINT := 16#0A57;   // f64,  bidir
    DP_ID_LEVI_KI_YAW_INITIAL                : UINT := 16#0A58;   // f64,  bidir

    DP_ID_PROP_FLAG                          : UINT := 16#0B00;   // u8,  bidir,  critical
    DP_ID_PROP_POSITION                      : UINT := 16#0B01;   // f64,  m,  pod->gs
    DP_ID_PROP_POSITION_INTERPOLATED         : UINT := 16#0B02;   // f64,  m,  pod->gs
    DP_ID_PROP_VELOCITY                      : UINT := 16#0B03;   // f64,  mm/s,  pod->gs
    DP_ID_PROP_FAULT_RIGHT                   : UINT := 16#0B04;   // u16,  pod->gs,  critical
    DP_ID_PROP_FAULT_LEFT                    : UINT := 16#0B05;   // u16,  pod->gs,  critical
    DP_ID_PROP_CURRENT_ANGLE_RIGHT           : UINT := 16#0B06;   // f64,  deg,  pod->gs
    DP_ID_PROP_CURRENT_ANGLE_LEFT            : UINT := 16#0B07;   // f64,  deg,  pod->gs
    DP_ID_PROP_TARGET_VELOCITY               : UINT := 16#0B08;   // i32,  mm/s,  bidir,  critical
    DP_ID_PROP_V_BUS_RIGHT                   : UINT := 16#0B09;   // f64,  V,  pod->gs
    DP_ID_PROP_V_BUS_LEFT                    : UINT := 16#0B0A;   // f64,  V,  pod->gs
    DP_ID_PROP_STATE_RIGHT                   : UINT := 16#0B0B;   // u16,  pod->gs
    DP_ID_PROP_STATE_LEFT                    : UINT := 16#0B0C;   // u16,  pod->gs
    DP_ID_PROP_ID_RIGHT                      : UINT := 16#0B0D;   // f64,  A,  pod->gs
    DP_ID_PROP_IQ_RIGHT                      : UINT := 16#0B0E;   // f64,  A,  pod->gs
    DP_ID_PROP_IA_RIGHT                      : UINT := 16#0B0F;   // f64,  A,  pod->gs
    DP_ID_PROP_IB_RIGHT                      : UINT := 16#0B10;   // f64,  A,  pod->gs
    DP_ID_PROP_IC_RIGHT                      : UINT := 16#0B11;   // f64,  A,  pod->gs
    DP_ID_PROP_ID_LEFT                       : UINT := 16#0B12;   // f64,  A,  pod->gs
    DP_ID_PROP_IQ_LEFT                       : UINT := 16#0B13;   // f64,  A,  pod->gs
    DP_ID_PROP_IA_LEFT                       : UINT := 16#0B14;   // f64,  A,  pod->gs
    DP_ID_PROP_IB_LEFT                       : UINT := 16#0B15;   // f64,  A,  pod->gs
    DP_ID_PROP_IC_LEFT                       : UINT := 16#0B16;   // f64,  A,  pod->gs
    DP_ID_PROP_DRIVE_RESET                   : UINT := 16#0B17;   // u8,  bidir,  critical
    DP_ID_PROP_AUTO_PILOT_FLAG               : UINT := 16#0B18;   // u8,  bidir,  critical
    DP_ID_PROP_TA_GD_LEFT                    : UINT := 16#0B19;   // u16,  deci-degC,  pod->gs
    DP_ID_PROP_TB_GD_LEFT                    : UINT := 16#0B1A;   // u16,  deci-degC,  pod->gs
    DP_ID_PROP_TC_GD_LEFT                    : UINT := 16#0B1B;   // u16,  deci-degC,  pod->gs
    DP_ID_PROP_TA_GD_RIGHT                   : UINT := 16#0B1C;   // u16,  deci-degC,  pod->gs
    DP_ID_PROP_TB_GD_RIGHT                   : UINT := 16#0B1D;   // u16,  deci-degC,  pod->gs
    DP_ID_PROP_TC_GD_RIGHT                   : UINT := 16#0B1E;   // u16,  deci-degC,  pod->gs
    DP_ID_PROP_POSITION_LIMIT_LOW            : UINT := 16#0B1F;   // u32,  m,  bidir
    DP_ID_PROP_POSITION_LIMIT_HIGH           : UINT := 16#0B20;   // u32,  m,  bidir
    DP_ID_PROP_MAX_THRUST                    : UINT := 16#0B21;   // u32,  N,  bidir

    DP_ID_TEMP_LEVI_FL1                      : UINT := 16#0C00;   // i32,  degC,  pod->gs,  critical
    DP_ID_TEMP_LEVI_FL2                      : UINT := 16#0C01;   // i32,  degC,  pod->gs,  critical
    DP_ID_TEMP_LEVI_FR1                      : UINT := 16#0C02;   // i32,  degC,  pod->gs,  critical
    DP_ID_TEMP_LEVI_FR2                      : UINT := 16#0C03;   // i32,  degC,  pod->gs,  critical
    DP_ID_TEMP_LEVI_BL1                      : UINT := 16#0C04;   // i32,  degC,  pod->gs,  critical
    DP_ID_TEMP_LEVI_BL2                      : UINT := 16#0C05;   // i32,  degC,  pod->gs,  critical
    DP_ID_TEMP_LEVI_BR1                      : UINT := 16#0C06;   // i32,  degC,  pod->gs,  critical
    DP_ID_TEMP_LEVI_BR2                      : UINT := 16#0C07;   // i32,  degC,  pod->gs,  critical
    DP_ID_TEMP_PROP_FL1                      : UINT := 16#0C08;   // i32,  degC,  pod->gs,  critical
    DP_ID_TEMP_PROP_FL2                      : UINT := 16#0C09;   // i32,  degC,  pod->gs,  critical
    DP_ID_TEMP_PROP_FL3                      : UINT := 16#0C0A;   // i32,  degC,  pod->gs,  critical
    DP_ID_TEMP_PROP_FL4                      : UINT := 16#0C0B;   // i32,  degC,  pod->gs,  critical
    DP_ID_TEMP_PROP_FR1                      : UINT := 16#0C0C;   // i32,  degC,  pod->gs,  critical
    DP_ID_TEMP_PROP_FR2                      : UINT := 16#0C0D;   // i32,  degC,  pod->gs,  critical
    DP_ID_TEMP_PROP_FR3                      : UINT := 16#0C0E;   // i32,  degC,  pod->gs,  critical
    DP_ID_TEMP_PROP_FR4                      : UINT := 16#0C0F;   // i32,  degC,  pod->gs,  critical
    DP_ID_TEMP_PROP_BL1                      : UINT := 16#0C10;   // i32,  degC,  pod->gs,  critical
    DP_ID_TEMP_PROP_BL2                      : UINT := 16#0C11;   // i32,  degC,  pod->gs,  critical
    DP_ID_TEMP_PROP_BL3                      : UINT := 16#0C12;   // i32,  degC,  pod->gs,  critical
    DP_ID_TEMP_PROP_BL4                      : UINT := 16#0C13;   // i32,  degC,  pod->gs,  critical
    DP_ID_TEMP_PROP_BR1                      : UINT := 16#0C14;   // i32,  degC,  pod->gs,  critical
    DP_ID_TEMP_PROP_BR2                      : UINT := 16#0C15;   // i32,  degC,  pod->gs,  critical
    DP_ID_TEMP_PROP_BR3                      : UINT := 16#0C16;   // i32,  degC,  pod->gs,  critical
    DP_ID_TEMP_PROP_BR4                      : UINT := 16#0C17;   // i32,  degC,  pod->gs,  critical
    DP_ID_TEMP_PROP_LOOP_IN                  : UINT := 16#0C18;   // i32,  degC,  pod->gs,  critical
    DP_ID_TEMP_PROP_LOOP_OUT                 : UINT := 16#0C19;   // i32,  degC,  pod->gs,  critical
    DP_ID_TEMP_LEVI_LOOP_IN                  : UINT := 16#0C1A;   // i32,  degC,  pod->gs,  critical
    DP_ID_TEMP_LEVI_LOOP_OUT                 : UINT := 16#0C1B;   // i32,  degC,  pod->gs,  critical
    DP_ID_FLOW_LEVI_FL                       : UINT := 16#0C1C;   // i32,  pod->gs
    DP_ID_FLOW_LEVI_FR                       : UINT := 16#0C1D;   // i32,  pod->gs
    DP_ID_FLOW_LEVI_BL                       : UINT := 16#0C1E;   // i32,  pod->gs
    DP_ID_FLOW_LEVI_BR                       : UINT := 16#0C1F;   // i32,  pod->gs
    DP_ID_FLOW_PROP_L1                       : UINT := 16#0C20;   // i32,  pod->gs
    DP_ID_FLOW_PROP_L2                       : UINT := 16#0C21;   // i32,  pod->gs
    DP_ID_FLOW_PROP_L3                       : UINT := 16#0C22;   // i32,  pod->gs
    DP_ID_FLOW_PROP_L4                       : UINT := 16#0C23;   // i32,  pod->gs
    DP_ID_FLOW_PROP_L5                       : UINT := 16#0C24;   // i32,  pod->gs
    DP_ID_FLOW_PROP_L6                       : UINT := 16#0C25;   // i32,  pod->gs
    DP_ID_FLOW_PROP_R1                       : UINT := 16#0C26;   // i32,  pod->gs
    DP_ID_FLOW_PROP_R2                       : UINT := 16#0C27;   // i32,  pod->gs
    DP_ID_FLOW_PROP_R3                       : UINT := 16#0C28;   // i32,  pod->gs
    DP_ID_FLOW_PROP_R4                       : UINT := 16#0C29;   // i32,  pod->gs
    DP_ID_FLOW_PROP_R5                       : UINT := 16#0C2A;   // i32,  pod->gs
    DP_ID_FLOW_PROP_R6                       : UINT := 16#0C2B;   // i32,  pod->gs
    DP_ID_THERM_EMS0                         : UINT := 16#0C2C;   // f32,  degC,  pod->gs,  critical
    DP_ID_THERM_EMS1                         : UINT := 16#0C2D;   // f32,  degC,  pod->gs,  critical
    DP_ID_THERM_EMS2                         : UINT := 16#0C2E;   // f32,  degC,  pod->gs,  critical
    DP_ID_THERM_EMS3                         : UINT := 16#0C2F;   // f32,  degC,  pod->gs,  critical
    DP_ID_THERM_EMS4                         : UINT := 16#0C30;   // f32,  degC,  pod->gs,  critical
    DP_ID_THERM_EMS5                         : UINT := 16#0C31;   // f32,  degC,  pod->gs,  critical
    DP_ID_THERM_EMS6                         : UINT := 16#0C32;   // f32,  degC,  pod->gs,  critical
    DP_ID_THERM_EMS7                         : UINT := 16#0C33;   // f32,  degC,  pod->gs,  critical
    DP_ID_THERM_HEMS0                        : UINT := 16#0C34;   // f32,  degC,  pod->gs,  critical
    DP_ID_THERM_HEMS1                        : UINT := 16#0C35;   // f32,  degC,  pod->gs,  critical
    DP_ID_THERM_HEMS2                        : UINT := 16#0C36;   // f32,  degC,  pod->gs,  critical
    DP_ID_THERM_HEMS3                        : UINT := 16#0C37;   // f32,  degC,  pod->gs,  critical
    DP_ID_THERM_HEMS4                        : UINT := 16#0C38;   // f32,  degC,  pod->gs,  critical
    DP_ID_THERM_HEMS5                        : UINT := 16#0C39;   // f32,  degC,  pod->gs,  critical
    DP_ID_THERM_HEMS6                        : UINT := 16#0C3A;   // f32,  degC,  pod->gs,  critical
    DP_ID_THERM_HEMS7                        : UINT := 16#0C3B;   // f32,  degC,  pod->gs,  critical
    DP_ID_THERM_MOTOR_LEFT_FRONT_0           : UINT := 16#0C3C;   // f32,  degC,  pod->gs,  critical
    DP_ID_THERM_MOTOR_LEFT_FRONT_1           : UINT := 16#0C3D;   // f32,  degC,  pod->gs,  critical
    DP_ID_THERM_MOTOR_LEFT_FRONT_2           : UINT := 16#0C3E;   // f32,  degC,  pod->gs,  critical
    DP_ID_THERM_MOTOR_LEFT_FRONT_3           : UINT := 16#0C3F;   // f32,  degC,  pod->gs,  critical
    DP_ID_THERM_MOTOR_LEFT_FRONT_4           : UINT := 16#0C40;   // f32,  degC,  pod->gs,  critical
    DP_ID_THERM_MOTOR_LEFT_FRONT_5           : UINT := 16#0C41;   // f32,  degC,  pod->gs,  critical
    DP_ID_THERM_MOTOR_LEFT_FRONT_6           : UINT := 16#0C42;   // f32,  degC,  pod->gs,  critical
    DP_ID_THERM_MOTOR_LEFT_FRONT_7           : UINT := 16#0C43;   // f32,  degC,  pod->gs,  critical
    DP_ID_THERM_MOTOR_LEFT_FRONT_8           : UINT := 16#0C44;   // f32,  degC,  pod->gs,  critical
    DP_ID_THERM_MOTOR_RIGHT_FRONT_0          : UINT := 16#0C45;   // f32,  degC,  pod->gs,  critical
    DP_ID_THERM_MOTOR_RIGHT_FRONT_1          : UINT := 16#0C46;   // f32,  degC,  pod->gs,  critical
    DP_ID_THERM_MOTOR_RIGHT_FRONT_2          : UINT := 16#0C47;   // f32,  degC,  pod->gs,  critical
    DP_ID_THERM_MOTOR_RIGHT_FRONT_3          : UINT := 16#0C48;   // f32,  degC,  pod->gs,  critical
    DP_ID_THERM_MOTOR_RIGHT_FRONT_4          : UINT := 16#0C49;   // f32,  degC,  pod->gs,  critical
    DP_ID_THERM_MOTOR_RIGHT_FRONT_5          : UINT := 16#0C4A;   // f32,  degC,  pod->gs,  critical
    DP_ID_THERM_MOTOR_RIGHT_FRONT_6          : UINT := 16#0C4B;   // f32,  degC,  pod->gs,  critical
    DP_ID_THERM_MOTOR_RIGHT_FRONT_7          : UINT := 16#0C4C;   // f32,  degC,  pod->gs,  critical
    DP_ID_THERM_MOTOR_RIGHT_FRONT_8          : UINT := 16#0C4D;   // f32,  degC,  pod->gs,  critical
    DP_ID_THERM_MOTOR_LEFT_BACK_0            : UINT := 16#0C4E;   // f32,  degC,  pod->gs,  critical
    DP_ID_THERM_MOTOR_LEFT_BACK_1            : UINT := 16#0C4F;   // f32,  degC,  pod->gs,  critical
    DP_ID_THERM_MOTOR_LEFT_BACK_2            : UINT := 16#0C50;   // f32,  degC,  pod->gs,  critical
    DP_ID_THERM_MOTOR_LEFT_BACK_3            : UINT := 16#0C51;   // f32,  degC,  pod->gs,  critical
    DP_ID_THERM_MOTOR_LEFT_BACK_4            : UINT := 16#0C52;   // f32,  degC,  pod->gs,  critical
    DP_ID_THERM_MOTOR_LEFT_BACK_5            : UINT := 16#0C53;   // f32,  degC,  pod->gs,  critical
    DP_ID_THERM_MOTOR_LEFT_BACK_6            : UINT := 16#0C54;   // f32,  degC,  pod->gs,  critical
    DP_ID_THERM_MOTOR_LEFT_BACK_7            : UINT := 16#0C55;   // f32,  degC,  pod->gs,  critical
    DP_ID_THERM_MOTOR_LEFT_BACK_8            : UINT := 16#0C56;   // f32,  degC,  pod->gs,  critical
    DP_ID_THERM_MOTOR_RIGHT_BACK_0           : UINT := 16#0C57;   // f32,  degC,  pod->gs,  critical
    DP_ID_THERM_MOTOR_RIGHT_BACK_1           : UINT := 16#0C58;   // f32,  degC,  pod->gs,  critical
    DP_ID_THERM_MOTOR_RIGHT_BACK_2           : UINT := 16#0C59;   // f32,  degC,  pod->gs,  critical
    DP_ID_THERM_MOTOR_RIGHT_BACK_3           : UINT := 16#0C5A;   // f32,  degC,  pod->gs,  critical
    DP_ID_THERM_MOTOR_RIGHT_BACK_4           : UINT := 16#0C5B;   // f32,  degC,  pod->gs,  critical
    DP_ID_THERM_MOTOR_RIGHT_BACK_5           : UINT := 16#0C5C;   // f32,  degC,  pod->gs,  critical
    DP_ID_THERM_MOTOR_RIGHT_BACK_6           : UINT := 16#0C5D;   // f32,  degC,  pod->gs,  critical
    DP_ID_THERM_MOTOR_RIGHT_BACK_7           : UINT := 16#0C5E;   // f32,  degC,  pod->gs,  critical
    DP_ID_THERM_MOTOR_RIGHT_BACK_8           : UINT := 16#0C5F;   // f32,  degC,  pod->gs,  critical
    DP_ID_THERM_FLOW_0                       : UINT := 16#0C60;   // f32,  degC,  pod->gs,  critical
    DP_ID_THERM_FLOW_1                       : UINT := 16#0C61;   // f32,  degC,  pod->gs,  critical
    DP_ID_THERM_FLOW_2                       : UINT := 16#0C62;   // f32,  degC,  pod->gs,  critical
    DP_ID_THERM_FLOW_3                       : UINT := 16#0C63;   // f32,  degC,  pod->gs,  critical
    DP_ID_THERM_FLOW_4                       : UINT := 16#0C64;   // f32,  degC,  pod->gs,  critical
    DP_ID_THERM_FLOW_5                       : UINT := 16#0C65;   // f32,  degC,  pod->gs,  critical
    DP_ID_THERM_FLOW_6                       : UINT := 16#0C66;   // f32,  degC,  pod->gs,  critical
    DP_ID_THERM_FLOW_7                       : UINT := 16#0C67;   // f32,  degC,  pod->gs,  critical
    DP_ID_FLOW_ARRAY_0                       : UINT := 16#0C68;   // f32,  pod->gs
    DP_ID_FLOW_ARRAY_1                       : UINT := 16#0C69;   // f32,  pod->gs
    DP_ID_FLOW_ARRAY_2                       : UINT := 16#0C6A;   // f32,  pod->gs
    DP_ID_FLOW_ARRAY_3                       : UINT := 16#0C6B;   // f32,  pod->gs
    DP_ID_FLOW_ARRAY_4                       : UINT := 16#0C6C;   // f32,  pod->gs
    DP_ID_FLOW_ARRAY_5                       : UINT := 16#0C6D;   // f32,  pod->gs
    DP_ID_FLOW_ARRAY_6                       : UINT := 16#0C6E;   // f32,  pod->gs
    DP_ID_FLOW_ARRAY_7                       : UINT := 16#0C6F;   // f32,  pod->gs
    DP_ID_FLOW_ARRAY_8                       : UINT := 16#0C70;   // f32,  pod->gs
    DP_ID_FLOW_ARRAY_9                       : UINT := 16#0C71;   // f32,  pod->gs
    DP_ID_OVERHEAT_HEMS                      : UINT := 16#0C72;   // u8,  pod->gs,  critical
    DP_ID_OVERHEAT_EMS                       : UINT := 16#0C73;   // u8,  pod->gs,  critical
    DP_ID_OVERHEAT_MOTOR                     : UINT := 16#0C74;   // u8,  pod->gs,  critical
    DP_ID_OVERHEAT_FLOW                      : UINT := 16#0C75;   // u8,  pod->gs,  critical
    DP_ID_PROP_DUTY_CYCLE                    : UINT := 16#0C76;   // f32,  pod->gs

    DP_ID_PTC_STATE                          : UINT := 16#0D00;   // u16,  pod->gs,  critical
    DP_ID_HVAL_STATUS                        : UINT := 16#0D01;   // u16,  pod->gs
    DP_ID_IMD_WARNINGS                       : UINT := 16#0D02;   // u16,  pod->gs
    DP_ID_PT_ERROR_STATUS                    : UINT := 16#0D03;   // u16,  pod->gs,  critical
    DP_ID_PT_FAIL_REASON                     : UINT := 16#0D04;   // u16,  pod->gs,  critical
    DP_ID_ISO_RES                            : UINT := 16#0D05;   // u32,  kOhm,  pod->gs,  critical
    DP_ID_IVT_CURRENT                        : UINT := 16#0D06;   // i32,  pod->gs,  critical
    DP_ID_PT_MAX_VOLTAGE                     : UINT := 16#0D07;   // u32,  pod->gs,  critical
    DP_ID_PT_MIN_VOLTAGE                     : UINT := 16#0D08;   // u32,  pod->gs,  critical
    DP_ID_PT_MAX_TEMP                        : UINT := 16#0D09;   // u32,  pod->gs,  critical
    DP_ID_PT_MIN_TEMP                        : UINT := 16#0D0A;   // u32,  pod->gs,  critical
    DP_ID_PT_TOTAL_VOLTAGE                   : UINT := 16#0D0B;   // u32,  pod->gs,  critical
    DP_ID_PT_PACK_CURRENT                    : UINT := 16#0D0C;   // u32,  pod->gs,  critical
    DP_ID_PTDC_LINK_VOLTAGE                  : UINT := 16#0D0D;   // i32,  pod->gs,  critical
	
	DP_ID_PT_LVSOC							: UINT := 16#0D0E;
	DP_ID_PT_LVVOLT							: UINT := 16#0D0F;
	DP_ID_PT_LVCUR							: UINT := 16#0D10;
	DP_ID_PT_LVTEMP							: UINT := 16#0D11;
	
	DP_ID_PT_HVSOC							: UINT := 16#0D12;
	

    DP_ID_CAN_LOG                            : UINT := 16#0FFD;
END_VAR

(* stored: Version 1.1.0.1
   GVL GVL_GS_IDS: Id {d6d88c6c-2e05-4e25-8922-249ed3619dac} *)
